FUNCTION_BLOCK SECOND_ORDER_SYSTEM (* 2nd ordem system y'' + K2y' + K1y = K*Xin *)
  (* Standard: 61499-2 *)
  (* Version 11-01-12, GASR *)
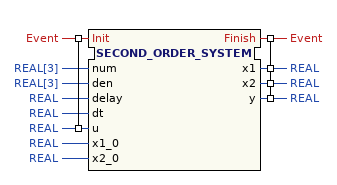
  EVENT_INPUT
    Init WITH u;
  END_EVENT
  EVENT_OUTPUT
    Finish WITH x1, x2, y;
  END_EVENT
  VAR_INPUT
    num : ARRAY [0..2] OF REAL;
    den : ARRAY [0..2] OF REAL;
    delay : REAL := 0;
    dt : REAL;
    u : REAL;
    x1_0 : REAL; (* condicao inicial *)
    x2_0 : REAL;
  END_VAR
  VAR_OUTPUT
    x1 : REAL;
    x2 : REAL;
    y : REAL;
  END_VAR
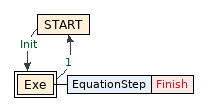
  EC_STATES
    Exe : EquationStep -> Finish;
    START;
  END_STATES
  EC_TRANSITIONS
    Exe TO START := 1;
    START TO Exe := Init;
  END_TRANSITIONS
  ALGORITHM EquationStep IN Lua: (* den[1] = b0, den[2] = b1 *)

						if type(input_buffer) ~= 'table' then
							input_buffer = {}
							for i = 1, math.ceil(delay/dt) +2 do
								input_buffer[#input_buffer +1] = 0
							end
						end
						input_buffer[#input_buffer] = u
						u = input_buffer[1]
						for i = 1, #input_buffer-1 do
							input_buffer[i] = input_buffer[i+1]
						end
						local beta1 = (num[2] - den[2]*num[1])
						local beta2 = num[3] - den[2]*beta1 - num[1]*den[3];

						local function f1(X1, X2, U)
							return X2 + beta1*U
						end

						local function f2(X1, X2, U)
							return (-den[3]*X1 - den[2]*X2 + beta2*U)
						end

						R11 = dt*f1(x1_0, x2_0, u);
						R12 = dt*f2(x1_0, x2_0, u);

						x1aux = x1_0 + 0.5*R11
						x2aux = x2_0 + 0.5*R12

						R21 = dt*f1(x1aux, x2aux, u);
						R22 = dt*f2(x1aux, x2aux, u);

						x1aux = x1aux + 0.5*R21
						x2aux = x2aux + 0.5*R22

						R31 = dt*f1(x1aux, x2aux, u);
						R32 = dt*f2(x1aux, x2aux, u);

						x1aux = x1aux + 0.5*R31
						x2aux = x2aux + 0.5*R32

						R41 = dt*f1(x1aux, x2aux, u);
						R42 = dt*f2(x1aux, x2aux, u);


						x1 = x1_0 + (1/6)*(R11 + 2*R21 + 2*R31 + R41)
						x2 = x2_0 + (1/6)*(R12 + 2*R22 + 2*R32 + R42)


						y  = x1 + num[1]*u

						x1_0 = x1
						x2_0 = x2
  END_ALGORITHM
END_FUNCTION_BLOCK
(* other elements stored in the file *)
(* VarDeclaration Name=R11 Type=REAL *)
(* VarDeclaration Name=R12 Type=REAL *)
(* VarDeclaration Name=R21 Type=REAL *)
(* VarDeclaration Name=R22 Type=REAL *)
(* VarDeclaration Name=R31 Type=REAL *)
(* VarDeclaration Name=R32 Type=REAL *)
(* VarDeclaration Name=R41 Type=REAL *)
(* VarDeclaration Name=R42 Type=REAL *)
(* VarDeclaration Name=x1aux Type=REAL *)
(* VarDeclaration Name=x2aux Type=REAL *)
(* VarDeclaration Name=input_buffer Type=REAL *)
